(* PLC project  *)

CONFIGURATION FSOE_1
END_CONFIGURATION
